(* Logix 5000 project; controller AOI_Test_3 vendor 1 type 14 code 108 rev 28.12; software revision 28.02 *)

TASK MainTask (continuous, watchdog 500 ms) : MainProgram

MODULES
   Local : vendor 1 type 14 code 108 (Compact 0, rev 28.12)
END_MODULES

TYPE AcceptResponse :
STRUCT
   Instance : DINT;
   Addr : SockAddr;
END_STRUCT
END_TYPE

TYPE OpenConnParams :
STRUCT
   Timeout : DINT;
   DestAddr : STRING;
END_STRUCT
END_TYPE

TYPE ReadParams :
STRUCT
   Timeout : DINT;
   BufLen : DINT;
END_STRUCT
END_TYPE

TYPE ReadResponse :
STRUCT
   FromAddr : SockAddr;
   BufLen : DINT;
   Buf : SINT[480];
END_STRUCT
END_TYPE

TYPE send :
STRUCT
   LEN : DINT;
   DATA : SINT[400];
END_STRUCT
END_TYPE

TYPE SockAddr :
STRUCT
   Family : INT;
   Port : INT;
   Addr : DINT;
END_STRUCT
END_TYPE

TYPE WriteParams :
STRUCT
   Timeout : DINT;
   ToAddr : SockAddr;
   BufLen : DINT;
   Buf : SINT[480];
END_STRUCT
END_TYPE

ADD_ON_INSTRUCTION TCP_Client_Comms   (* revision 1.0 *)
VAR_IN_OUT
   Delete_Sockets_All : MESSAGE; {required}
   Create_Socket : MESSAGE; {required}
   Socket_Open_Connection : MESSAGE; {required}
   Socket_Read : MESSAGE; {required}
   Socket_Write : MESSAGE; {required}
   so_CreateParams : AcceptResponse; {required}
   so_CreateInstance : DINT; {required}
   so_OpenParams : OpenConnParams; {required}
   so_ReadParams : ReadParams; {required}
   so_ReadResponse : ReadResponse; {required}
   so_WriteParams : WriteParams; {required}
   so_WriteResponse : DINT; {required}
END_VAR
VAR_INPUT
   Remote_Port : DINT := 21; {access None, required}
END_VAR
VAR_IN_OUT
   Remote_IP : STRING; {required}
   Write : STRING; {required}
   Read : STRING; {required}
   Reset : BOOL; {required}
END_VAR
VAR
   Port_Str : STRING; {access None}
   IP_PORT_SNDRD : STRING := '?port='; {access None}
   Timeout : DINT := 1000; {access None}
   ONS_TCP : BOOL[32]; {access None}
   Create_Instance : DINT := 1; {access None}
   Create_Family : DINT := 2; {access None}
   Create_Port : DINT; {access None}
   Create_Address : DINT; {access None}
   Read_BufLen : DINT := 82; {access None}
   Read_Params_BufLen : DINT := 100; {access None}
   Write_Params_BufLen : DINT := 11; {access None}
   Write_Response : DINT := 216; {access None}
   Read_Write_Refresh_Delay : TIMER := (PRE := 2000); {access None}
   send : send; {access None}
   Data_Clear : DINT; {access None}
   Clear_Lock : BOOL; {access None}
   Done_Write_Clear : BOOL; {access None}
   numchars : DINT; {access None}
   Null_String : STRING; {access None}
END_VAR

ROUTINE Logic   (* ladder *)
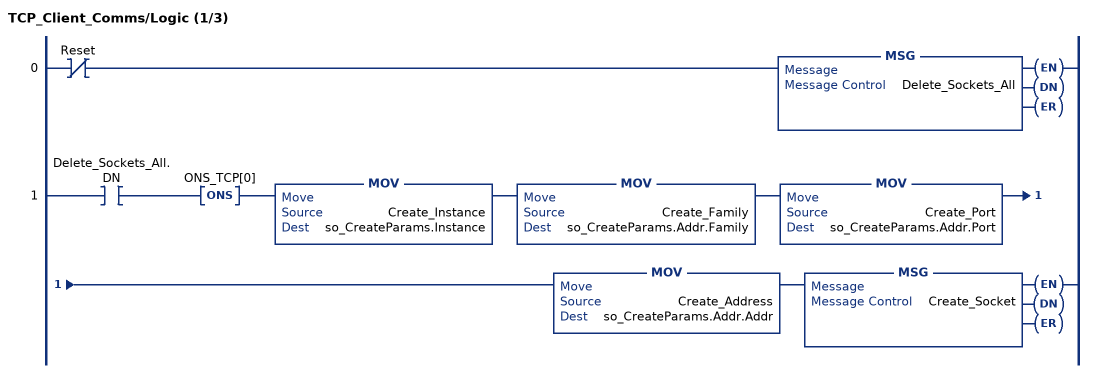
   0: XIO(Reset)MSG(Delete_Sockets_All);
   1: XIC(Delete_Sockets_All.DN)ONS(ONS_TCP[0])MOV(Create_Instance,so_CreateParams.Instance)MOV(Create_Family,so_CreateParams.Addr.Family)MOV(Create_Port,so_CreateParams.Addr.Port)MOV(Create_Address,so_CreateParams.Addr.Addr)MSG(Create_Socket);
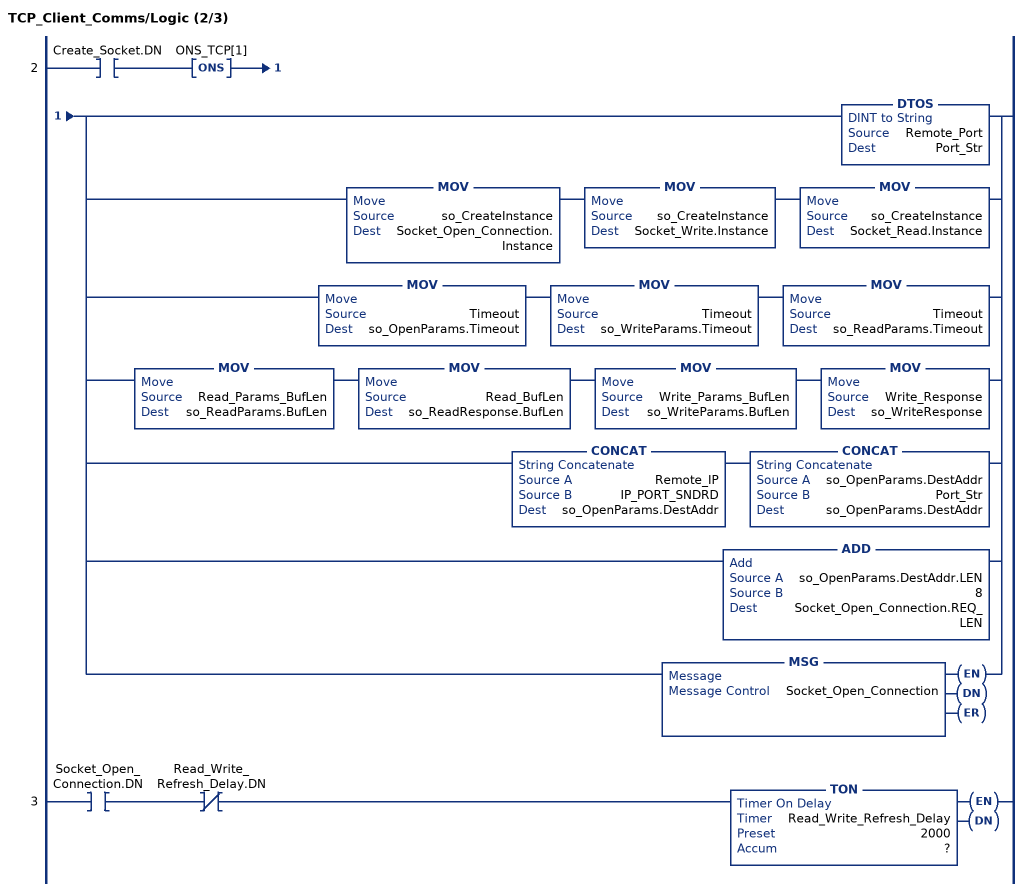
   2: XIC(Create_Socket.DN)ONS(ONS_TCP[1])[DTOS(Remote_Port,Port_Str) ,MOV(so_CreateInstance,Socket_Open_Connection.Instance) MOV(so_CreateInstance,Socket_Write.Instance) MOV(so_CreateInstance,Socket_Read.Instance) ,MOV(Timeout,so_OpenParams.Timeout) MOV(Timeout,so_WriteParams.Timeout) MOV(Timeout,so_ReadParams.Timeout) ,MOV(Read_Params_BufLen,so_ReadParams.BufLen) MOV(Read_BufLen,so_ReadResponse.BufLen) MOV(Write_Params_BufLen,so_WriteParams.BufLen) MOV(Write_Response,so_WriteResponse) ,CONCAT(Remote_IP,IP_PORT_SNDRD,so_OpenParams.DestAddr) CONCAT(so_OpenParams.DestAddr,Port_Str,so_OpenParams.DestAddr) ,ADD(so_OpenParams.DestAddr.LEN,8,Socket_Open_Connection.REQ_LEN) ,MSG(Socket_Open_Connection) ];
   3: XIC(Socket_Open_Connection.DN)XIO(Read_Write_Refresh_Delay.DN)TON(Read_Write_Refresh_Delay,?,?);
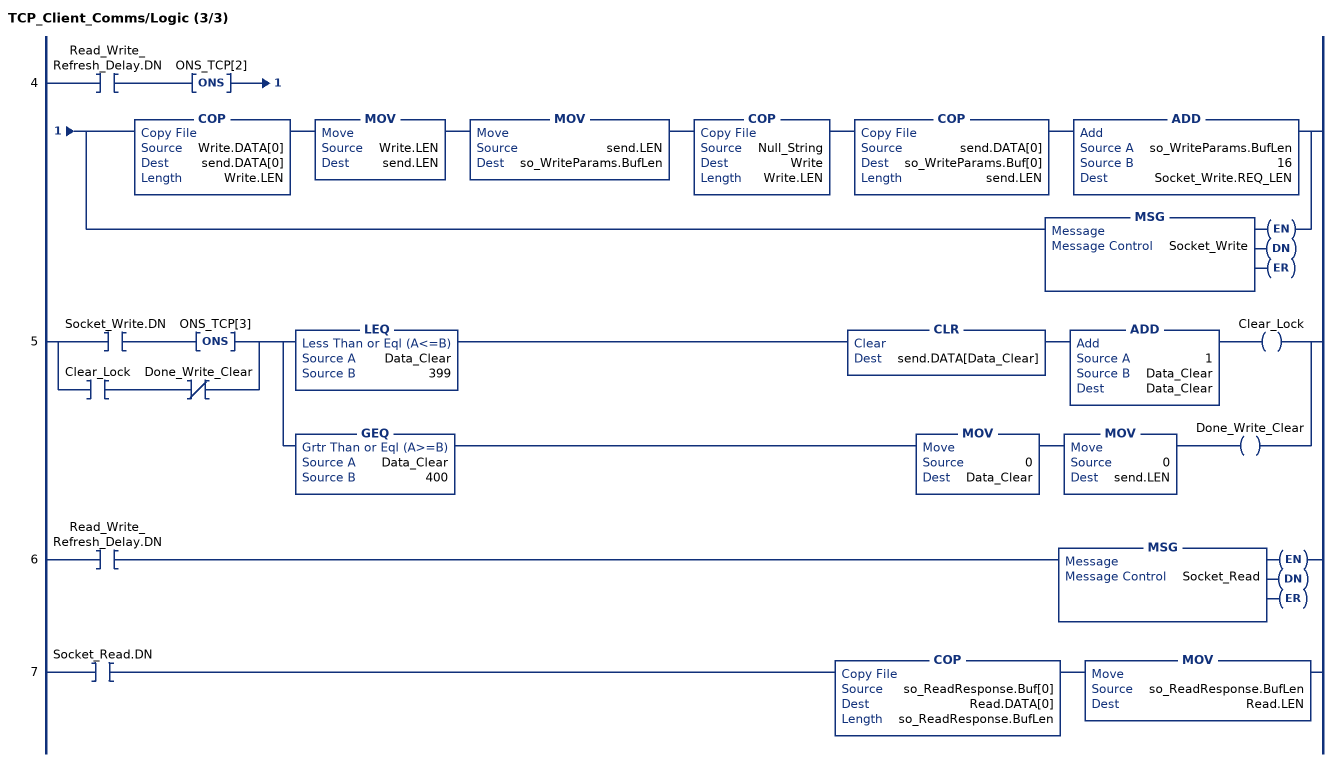
   4: XIC(Read_Write_Refresh_Delay.DN)ONS(ONS_TCP[2])[COP(Write.DATA[0],send.DATA[0],Write.LEN) MOV(Write.LEN,send.LEN) MOV(send.LEN,so_WriteParams.BufLen) COP(Null_String,Write,Write.LEN) COP(send.DATA[0],so_WriteParams.Buf[0],send.LEN) ADD(so_WriteParams.BufLen,16,Socket_Write.REQ_LEN) ,MSG(Socket_Write) ];
   5: [XIC(Socket_Write.DN) ONS(ONS_TCP[3]) ,XIC(Clear_Lock) XIO(Done_Write_Clear) ][LEQ(Data_Clear,399) CLR(send.DATA[Data_Clear]) ADD(1,Data_Clear,Data_Clear) OTE(Clear_Lock) ,GEQ(Data_Clear,400) MOV(0,Data_Clear) MOV(0,send.LEN) OTE(Done_Write_Clear) ];
   6: XIC(Read_Write_Refresh_Delay.DN)MSG(Socket_Read);
   7: XIC(Socket_Read.DN)COP(so_ReadResponse.Buf[0],Read.DATA[0],so_ReadResponse.BufLen)MOV(so_ReadResponse.BufLen,Read.LEN);
END_ROUTINE
END_ADD_ON_INSTRUCTION

VAR_GLOBAL   (* controller tags *)
   Create_Socket : MESSAGE;
        MessageParameters(ServiceCode := 16#004b, LocalElement := CreateParams, DestinationTag := CreateInstance, ...)
   CreateInstance : DINT := 17545;
   CreateParams : AcceptResponse := (Instance := 1, Addr.Family := 2);
   Delete_Sockets_All : MESSAGE;
        MessageParameters(ServiceCode := 16#0051, ...)
   OpenParams : OpenConnParams := (Timeout := 1000, DestAddr := '192.168.1.250?port=62');
   port : DINT := 62;
   Read : STRING;
   ReadParams : ReadParams := (Timeout := 1000, BufLen := 100);
   ReadResponse : ReadResponse := (Buf[0] := 104, Buf[1] := 105, Buf[2] := 13, Buf[3] := 10, Buf[4] := 111, Buf[5] := 32, Buf[6] := 119, Buf[7] := 111, Buf[8] := 114, Buf[9] := 108, Buf[10] := 100, Buf[11] := 13, Buf[12] := 10, Buf[13] := 10);
   Remote_IP : STRING := '192.168.1.250';
   Reset : BOOL;
   Socket_Open_Connection : MESSAGE;
        MessageParameters(ServiceCode := 16#004c, LocalElement := OpenParams, ...)
   Socket_Read : MESSAGE;
        MessageParameters(ServiceCode := 16#004d, LocalElement := ReadParams, DestinationTag := ReadResponse, ...)
   Socket_Write : MESSAGE;
        MessageParameters(ServiceCode := 16#004e, LocalElement := WriteParams, DestinationTag := WriteResponse, ...)
   TCP_Client_Comms : TCP_Client_Comms := (Remote_Port := 62);
   toggle : BOOL := 1;
   Write : STRING;
   WriteParams : WriteParams := (Timeout := 1000, Buf[0] := 104, Buf[1] := 101, Buf[2] := 108, Buf[3] := 108, Buf[4] := 111, Buf[5] := 32, Buf[6] := 32, Buf[7] := 119, Buf[8] := 111, Buf[9] := 114, Buf[10] := 108, Buf[11] := 100);
   WriteResponse : DINT := 12;
END_VAR

PROGRAM MainProgram   (* main routine MainRoutine *)

ROUTINE MainRoutine   (* ladder *)
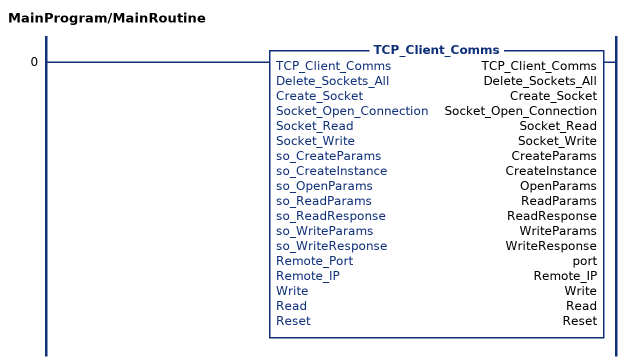
   0: TCP_Client_Comms(TCP_Client_Comms,Delete_Sockets_All,Create_Socket,Socket_Open_Connection,Socket_Read,Socket_Write,CreateParams,CreateInstance,OpenParams,ReadParams,ReadResponse,WriteParams,WriteResponse,port,Remote_IP,Write,Read,Reset);
END_ROUTINE
END_PROGRAM
